DATA_BLOCK "MotorControl"
VAR
  Dev : Array[1..20] of "Motor_Control";
END_VAR
BEGIN
END_DATA_BLOCK
